Fanuc KAREL source: kc00023.KL

-- PROVISIONAL review KL for V940-1; original PC SHA256 4527c097128fed54d572c98a2223463a3c31a5091b46237fca07d822c69314a6
-- Incomplete behavior may be omitted. Consult companion uncertainty JSON. Do not deploy.
PROGRAM KC00023
%NOLOCKGROUP
BEGIN
  -- V9_ZERO_TABLE_METADATA_HINT layout=0001; no indexed target words; source/name/runtime held
  -- UNRESOLVED_PC offsets 0-1; opcodes 7B
  -- UNRESOLVED_PC offsets 6-20; opcodes 2D,9D,52,2F
  -- UNRESOLVED_PC offsets 25-29; opcodes 7F
  -- UNRESOLVED_PC offsets 34-42; opcodes 3F,75
  -- UNRESOLVED_PC offsets 47-56; opcodes 3F,75
  -- UNRESOLVED_PC offsets 61-88; opcodes 27,73,73,22,24,AA,26
  -- UNRESOLVED_PC offsets 93-97; opcodes 7F
END KC00023
